// TwinCAT 3 PLC project Tags
// Title: Tags
// Company: _
// Author: Krystian Lis et al.
// ProjectVersion: 1.0.0
// Description: Universal identification.
// ProgramVersion: 3.1.4026.9
// libraries:
//   Tc2_Standard, * (Beckhoff Automation GmbH)
//   Tc2_Utilities, * (Beckhoff Automation GmbH)
//   Calls, * (_)
//   Debug, * (_)
//   Domains, * (_)
//   Results, * (_)
//   Strings, * (_)
// project tree:
//   Tag/Base/ TagProxy.TcPOU, I_Tag.TcIO, I_Tagged.TcIO, Tag.TcPOU
//   Tag/Buffer/ TagBuffer.TcPOU
//   Tag/Cmp/ I_TagCmp.TcIO, TagCmp.TcPOU
//   Tag/Owner/ I_TagOwner.TcIO, TagOwner.TcPOU (not stored)

// ---- Tag/Base/I_Tag.TcIO
INTERFACE I_Tag EXTENDS Debug.I_Debug, Domains.I_Component

PROPERTY Cache : UDINT
GET
END_GET
END_PROPERTY

METHOD GetId : Strings.Str
VAR_INPUT
END_VAR
END_METHOD

METHOD Join : Results.Result
VAR_INPUT
	iOwner		: I_TagOwner;
	nCache		: UDINT;
END_VAR
END_METHOD

METHOD Leave : Results.Result
VAR_INPUT
	iOwner		: I_TagOwner;
END_VAR
END_METHOD

PROPERTY Option : Strings.Str
GET
END_GET
END_PROPERTY

PROPERTY Owner : I_TagOwner
GET
END_GET
END_PROPERTY

PROPERTY Self : I_Tag
GET
END_GET
END_PROPERTY

END_INTERFACE

// ---- Tag/Base/I_Tagged.TcIO
INTERFACE I_Tagged EXTENDS Domains.I_Component

PROPERTY Tag : I_Tag
GET
END_GET
END_PROPERTY

END_INTERFACE

// ---- Tag/Cmp/I_TagCmp.TcIO
INTERFACE INTERNAL I_TagCmp

METHOD AndIf : I_TagCmp
VAR_INPUT
	bCondition: BOOL;
END_VAR
END_METHOD

METHOD HasOption : I_TagCmp
VAR_INPUT
	sOption		: Strings.Str;
END_VAR
END_METHOD

METHOD IsErr : BOOL
END_METHOD

METHOD IsFalse : BOOL
END_METHOD

METHOD IsTrue : BOOL
END_METHOD

METHOD Match : I_TagCmp
VAR_INPUT
	iOther: I_Tag;
END_VAR
END_METHOD

METHOD MatchId : I_TagCmp
VAR_INPUT
	sIdToMatch		: Strings.Str;
END_VAR
END_METHOD

METHOD MatchWcdId : I_TagCmp
VAR_INPUT
	sPattern 			: Strings.Str;  					// Pattern with wildcards
END_VAR
END_METHOD

METHOD OrIf : I_TagCmp
VAR_INPUT
	bCondition: BOOL;
END_VAR
END_METHOD

METHOD Set : I_TagCmp
VAR_INPUT
	iBaseTag	: I_Tag;
END_VAR
END_METHOD

METHOD XorIf : I_TagCmp
VAR_INPUT
	bCondition: BOOL;
END_VAR
END_METHOD

END_INTERFACE

// ---- Tag/Owner/I_TagOwner.TcIO
INTERFACE INTERNAL I_TagOwner

END_INTERFACE

// ---- Tag/Base/TagProxy.TcPOU
FUNCTION_BLOCK TagProxy IMPLEMENTS Debug.I_Debug

//FB_Init is always available implicitly and it is used primarily for initialization.
//The return value is not evaluated. For a specific influence, you can also declare the
//methods explicitly and provide additional code there with the standard initialization
//code. You can evaluate the return value.
METHOD FB_Init: BOOL
VAR_INPUT
    bInitRetains: BOOL; // TRUE: the retain variables are initialized (reset warm / reset cold)
    bInCopyCode: BOOL;  // TRUE: the instance will be copied to the copy code afterward (online change)
	
	iTag			: I_Tag;
	refTag			: REFERENCE TO I_Tag;
END_VAR
IF NOT __ISVALIDREF(refTag) THEN
	Debug.DebugMsg(THIS^, ': Ref = 0!');
	RETURN;
END_IF

IF iTag = 0 THEN
	Debug.DebugMsg(THIS^, ': Itf = 0!');
	RETURN;
END_IF

IF refTag <> 0 THEN
	Debug.DebugMsg(THIS^, ': Ref itf should be unassigned!');
	RETURN;
END_IF

refTag := iTag;
END_METHOD

END_FUNCTION_BLOCK

// ---- Tag/Base/Tag.TcPOU
{attribute 'reflection'}
FUNCTION_BLOCK Tag IMPLEMENTS I_Tag
VAR
	{attribute 'instance-path'} 
    {attribute 'noinit'} 
	_sId			: Strings.Str;
	_nOptionPos		: USINT;
	_nOptionLen		: USINT;
	_nCache			: UDINT;
	_iOwner			: I_TagOwner;
END_VAR

PROPERTY Cache : UDINT
GET
Cache := _nCache;
END_GET
END_PROPERTY

METHOD FB_init : BOOL
VAR_INPUT
	bInitRetains : BOOL; // if TRUE, the retain variables are initialized (warm start / cold start)
	bInCopyCode : BOOL;  // if TRUE, the instance afterwards gets moved into the copy code (online change)
END_VAR
VAR
	i				: INT;
	_sChar			: Strings.Ch;
	
END_VAR
// Delete this name
FOR i := Tc2_Standard.LEN(_sId) TO 1 BY -1 DO
	IF Tc2_Standard.MID(_sId, 1, i) = '.' THEN
		_sId := Tc2_Standard.LEFT(_sId, i - 1);
		EXIT;
	END_IF
END_FOR

// Delete project name
FOR i := 1 TO Tc2_Standard.LEN(_sId) DO
	IF Tc2_Standard.MID(_sId, 1, i) = '.' THEN
		_sId := Tc2_Standard.DELETE(_sId, i, 1);
		EXIT;
	END_IF
END_FOR

// Delete plc name
FOR i := 1 TO Tc2_Standard.LEN(_sId) DO
	IF Tc2_Standard.MID(_sId, 1, i) = '.' THEN
		_sId := Tc2_Standard.DELETE(_sId, i, 1);
		EXIT;
	END_IF
END_FOR

// Replace '[' with '.' and remove ']' 
FOR i := 1 TO Tc2_Standard.LEN(_sId) DO
	_sChar := Tc2_Standard.MID(_sId, 1, i);
	IF _sChar = '[' THEN
		_sId := Tc2_Standard.REPLACE(_sId, '.', 1, i);
	ELSIF _sChar = ']' THEN
		_sId := Tc2_Standard.DELETE(_sId, 1, i);
	END_IF
END_FOR

_sId := Tc2_Utilities.F_ToLCase(_sID);
END_METHOD

METHOD GetId : Strings.Str
VAR_INPUT
END_VAR
IF _nOptionPos <> 0 THEN
	GetId := Tc2_Standard.DELETE(_sId, _nOptionLen + 1, _nOptionPos); 
ELSE
	GetId := _sId;
END_IF
END_METHOD

METHOD Join : Results.Result
VAR_INPUT
	iOwner		: I_TagOwner;
	nCache		: UDINT;
END_VAR
IF iOwner = 0 THEN
	Join := Results.Err.Itf0;
	RETURN;
END_IF

IF _iOwner <> 0 THEN
	Join := Results.Err.ItfEq;
	RETURN;
END_IF

_iOwner := iOwner;
_nCache := nCache;
Join := Results.Ok;
END_METHOD

METHOD Leave : Results.Result
VAR_INPUT
	iOwner		: I_TagOwner;
END_VAR
IF iOwner = 0 THEN
	Leave := Results.Err.Itf0;
	RETURN;
END_IF

IF _iOwner <> iOwner THEN
	Leave := Results.Err.ItfEq;
	RETURN;
END_IF

_iOwner := 0;
Leave := Results.Ok;
END_METHOD

PROPERTY Option : Strings.Str
GET
VAR
	i				: INT;
END_VAR
IF _nOptionPos <> 0 THEN
	Option := Tc2_Standard.DELETE(_sId, _nOptionPos, 1); 
ELSE
	Option := '';
END_IF
END_GET
SET
IF Option <> '' THEN
    _nOptionLen := INT_TO_USINT(Tc2_Standard.LEN(Option));    
    IF _nOptionPos <> 0 THEN
        _sId := Tc2_Standard.LEFT(_sId, _nOptionPos);
        _sId := Tc2_Standard.CONCAT(_sId, Option);
    ELSE
        // The option does not exist, so we append it
        _nOptionPos := INT_TO_USINT(Tc2_Standard.LEN(_sId) + 1);
        _sId := Tc2_Standard.CONCAT(_sId, '.');
        _sId := Tc2_Standard.CONCAT(_sId, Option);
    END_IF
ELSIF _nOptionPos <> 0 THEN
    _sId := Tc2_Standard.LEFT(_sId, _nOptionPos - 1);
    _nOptionPos := 0;
END_IF
END_SET
END_PROPERTY

PROPERTY Owner : I_TagOwner
GET
Owner := _iOwner;
END_GET
END_PROPERTY

PROPERTY Self : I_Tag
GET
Self := THIS^;
END_GET
END_PROPERTY

END_FUNCTION_BLOCK

// ---- Tag/Buffer/TagBuffer.TcPOU
FUNCTION_BLOCK TagBuffer
VAR_GENERIC CONSTANT
	nMax			: UDINT := 0;
END_VAR
VAR
	_iBuffer		: ARRAY[0..nMax] OF I_Tag;
	_nHead			: UDINT := 0;
	_nTail			: UDINT := 0;
	_nLen			: UDINT := 0;
END_VAR

METHOD Clear
VAR
	i	: UDINT := _nHead;
	c	: UDINT	:= 0;
END_VAR
WHILE c < _nLen DO
	_iBuffer[i] := 0;

	i := (i + 1) MOD nMax;
	c := c + 1;
END_WHILE;
END_METHOD

METHOD Has : BOOL
VAR_INPUT
	iTag	: I_Tag;
END_VAR
VAR
	i	: UDINT := _nHead;
	c	: UDINT	:= 0;
END_VAR
IF iTag = 0 THEN
	Has := FALSE;
	RETURN;
END_IF

WHILE c < _nLen DO
	IF _iBuffer[i] = iTag THEN
		Has := TRUE;
		EXIT;
	END_IF;

	i := (i + 1) MOD nMax;
	c := c + 1;
END_WHILE;
END_METHOD

METHOD Pop : Results.Result
VAR_OUTPUT
	iTag		: I_Tag;
END_VAR
IF _nHead = _nTail THEN
    Pop := Results.None;
    RETURN;
END_IF

iTag := _iBuffer[_nHead];
_iBuffer[_nHead] := 0;

_nHead := _nHead + 1;
_nLen := _nLen - 1;

IF _nHead > nMax THEN
    _nHead := 0;
END_IF

Pop := Results.Ok;
END_METHOD

METHOD Push : Results.Result
VAR_INPUT
	iTag			: I_Tag;
END_VAR
VAR
	_nNextTail 		: UDINT;
END_VAR
IF iTag = 0 THEN
	Push := Results.Err.Itf0;
	RETURN;
END_IF

_nNextTail := _nTail + 1;

IF _nNextTail > nMax THEN
    _nNextTail := 0;
END_IF

IF _nNextTail = _nHead THEN
    Push := Results.Err.Ovf; 
    RETURN;
END_IF

_nLen := _nLen + 1;
_iBuffer[_nTail] := iTag;
_nTail := _nNextTail;
Push := Results.Ok;
END_METHOD

END_FUNCTION_BLOCK

// ---- Tag/Cmp/TagCmp.TcPOU
FUNCTION_BLOCK TagCmp IMPLEMENTS I_TagCmp
VAR
	_iBaseTag		: I_Tag;
	_eResult		: Results.Result;
	_bLock			: BOOL;
END_VAR

PROPERTY PRIVATE _self : I_TagCmp
GET
VAR
	_this : I_TagCmp := THIS^;
END_VAR
_self := _this;
END_GET
END_PROPERTY

METHOD AndHasOption : I_TagCmp
VAR_INPUT
	sOption		: Strings.Str;
END_VAR
AndHasOption := _self;
sOption := Tc2_Utilities.F_ToLCase(sOption);

IF _bLock THEN
	RETURN;
END_IF

CASE _eResult OF
	Results.Ok,
	Results.None:
		IF _eResult = Results.Ok AND_THEN sOption <> '' AND_THEN _iBaseTag.Option = sOption THEN
			_eResult := Results.Ok;
		END_IF
END_CASE
END_METHOD

METHOD AndIf : I_TagCmp
VAR_INPUT
	bCondition: BOOL;
END_VAR
AndIf := _self;

IF _bLock THEN
	RETURN;
END_IF

IF _eResult = Results.Ok AND_THEN bCondition THEN
	_eResult := Results.Ok;
END_IF
END_METHOD

METHOD HasOption : I_TagCmp
VAR_INPUT
	sOption		: Strings.Str;
END_VAR
HasOption := _self;
sOption := Tc2_Utilities.F_ToLCase(sOption);

IF _bLock THEN
	RETURN;
END_IF

CASE _eResult OF
	Results.Ok,
	Results.None:
		IF sOption <> '' AND_THEN _iBaseTag.Option = sOption THEN
			_eResult := Results.Ok;
		END_IF
END_CASE
END_METHOD

METHOD IsErr : BOOL
IF _bLock THEN
	RETURN;
END_IF

IF _eResult >= 0 THEN
	RETURN;
END_IF

_bLock := TRUE;
IsErr := TRUE;
END_METHOD

METHOD IsFalse : BOOL
IF _bLock THEN
	RETURN;
END_IF

IF _eResult <> Results.None THEN
	RETURN;
END_IF

_bLock := TRUE;
IsFalse := TRUE;
END_METHOD

METHOD IsTrue : BOOL
IF _bLock THEN
	RETURN;
END_IF

IF _eResult <> Results.Ok THEN
	RETURN;
END_IF

_bLock := TRUE;
IsTrue := TRUE;
END_METHOD

METHOD Match : I_TagCmp
VAR_INPUT
	iOther: I_Tag;
END_VAR
Match := _self;

IF _bLock THEN
	RETURN;
END_IF

CASE _eResult OF
	Results.Ok,
	Results.None:
		IF iOther = _iBaseTag THEN
			_eResult := Results.Ok;
		END_IF
END_CASE
END_METHOD

METHOD MatchId : I_TagCmp
VAR_INPUT
	sIdToMatch		: Strings.Str;
END_VAR
MatchId := _self;
sIdToMatch := Tc2_Utilities.F_ToLCase(sIdToMatch);

IF _bLock THEN
	RETURN;
END_IF

CASE _eResult OF
	Results.Ok,
	Results.None:
		IF sIdToMatch <> '' AND_THEN (Tc2_Standard.RIGHT(_iBaseTag.GetId(), Tc2_Standard.LEN(sIdToMatch)) = sIdToMatch) THEN
			_eResult := Results.Ok;
		END_IF
END_CASE
END_METHOD

METHOD MatchWcdId : I_TagCmp
VAR_INPUT
	sPattern 			: Strings.Str;  					// Pattern with wildcards
END_VAR
VAR
	pttPath				: Strings.SymbolPath;
	pttSeg				: Strings.Str;
	pttPeek				: Strings.Str;
	addPath				: Strings.SymbolPath;
	addSeg				: Strings.Str;
END_VAR
MatchWcdId := _self;

// Check lock
IF _bLock THEN
	RETURN;
END_IF

// Check result state
CASE _eResult OF
	Results.Ok,
	Results.None:
		pttPath.Set(sPattern);
		addPath.Set(_iBaseTag.GetId());
		WHILE Results.IsOk(pttPath.Next(sSeg => pttSeg)) DO
		
			IF pttSeg = '*' THEN
				IF Results.IsOk(pttPath.Peek(sSeg => pttPeek)) THEN
					IF pttPeek = '*' THEN
						CONTINUE; // Skip redundant wildcard
					END_IF
				ELSE
					RETURN; // No more segments in the pattern, so it's a match
				END_IF
	
			ELSIF pttSeg <> '*' THEN
				pttPeek := '';
			END_IF
			
			WHILE Results.IsOk(addPath.Next(sSeg => addSeg)) DO
				IF pttPeek <> '' THEN
					IF pttPeek = addSeg THEN
						pttPath.Next();
						EXIT;
					ELSE
						CONTINUE;
					END_IF
				ELSIF pttSeg = addSeg THEN
					EXIT;
				ELSE
					RETURN;
				END_IF
			END_WHILE		
		END_WHILE
		
		IF Results.IsOk(addPath.Peek()) THEN
			RETURN;
		END_IF
		
		_eResult := Results.Ok;
END_CASE
END_METHOD

METHOD OrIf : I_TagCmp
VAR_INPUT
	bCondition: BOOL;
END_VAR
OrIf := _self;

IF _bLock THEN
	RETURN;
END_IF

IF _eResult = Results.Ok OR_ELSE bCondition THEN
	_eResult := Results.Ok;
END_IF
END_METHOD

METHOD Set : I_TagCmp
VAR_INPUT
	iBaseTag	: I_Tag;
END_VAR
_iBaseTag := iBaseTag;
_eResult := Results.None;
_bLock := FALSE;

IF iBaseTag = 0 THEN
	_eResult := Results.Err.Itf0;
END_IF

Set := _self;
END_METHOD

METHOD XorIf : I_TagCmp
VAR_INPUT
	bCondition: BOOL;
END_VAR
XorIf := _self;

IF _bLock THEN
	RETURN;
END_IF

IF _eResult = Results.Ok XOR bCondition THEN
	_eResult := Results.Ok;
END_IF
END_METHOD

END_FUNCTION_BLOCK
